(* CODESYS project CtaAppBmk_1.0.0.0.library
   Description: Bmk Library der CTA
   Version: 1.0.0.0
   Title: CtaAppBmk
   Author: SIS
   Company: CTA
   DocFormat: reStructuredText
   Placeholder: CtaAppBmk
   DefaultNamespace: CtaAppBmk
   CompiledLibraryCompatibilityVersion: CODESYS V3.5 SP16 Patch 3
   LanguageModelAttribute: qualified-access-only

Project tree, tasks and I/O mapping:
  libraries: CtaSysBase, 1.0.0.0 (CTA); TextListUtils, * (System); CtaVisSymbols, 1.0.0.0 (CTA); VisuSymbols, 4.5.0.0 (System)
  40 Visualizations/
    visualisation visObjInfoIntern
    visualisation visObjInfo
  30 Program Organization Units/
    function block fbBMK [ST]: proGetBMK, proGetAKS, proGetVendorDesignation, proGetCustomerDesignation, proGetObjectId, proNoBmkInList
  00000000-0000-0000-0000-000000000000|D:\CoDeSys\LibrariesV3\trunk\Intern\CAA\CAA Template\3.4.0.0 draft\Placeholder.xml
  00000000-0000-0000-0000-000000000000|D:\CoDeSys\LibrariesV3\trunk\Intern\CAA\CAA Template\3.2.0.3 draft\Prefix.pdf
  00000000-0000-0000-0000-000000000000|D:\CoDeSys\LibrariesV3\trunk\Intern\CAA\CAA Template\3.5.2.0 draft\Placeholder.xml
  20 Structs/
  50 Images/
  10 Documenation/
    global variables VersionHistory
    global variables readMe
  21 Interface/
    interface ITF_BMK: proGetAKS, proGetBMK, proGetObjectId, proNoBmkInList, proGetCustomerDesignation, proGetVendorDesignation
  11 Library Parameter/
    global variables Parameter
  12 Konstanten/
  60 Textlisten/
  13 Globale Variablen/
  text list GlobalTextList
*)

// 10 Documenation/VersionHistory
(* 

.. image:: ../../Images/CTA_Logo.jpg
   :align: right
   :width: 15% 

**Vorlage**   


============ =========== =========== ============================================
**Date**     **Version** **Author**  **Change**
------------ ----------- ----------- --------------------------------------------
04.03.2021   0.0.0.0     SIS         Vorlage erstellt

============ =========== =========== ============================================


*)
VAR_GLOBAL
    stInfo : STRING:= '0.0.0.0, Vorlage, CTA';
END_VAR

// 10 Documenation/readMe
(*

**ReadMe**
 
 |	**Empfehlung**
 |
 |	Dokumentrieren Sie die Library für eine nachhaltige Entwicklung
 |     
 | *Beispiel* 
 |
 | Dies ist die Vorlage Library der CTA. Erstellen Sie ihre Library anhand dieser Vorlage.
*)

VAR_GLOBAL
    xReadMeDone              :   BOOL;
END_VAR

// 11 Library Parameter/Parameter
{attribute 'qualified_only' := ''}
VAR_GLOBAL CONSTANT
	stTextListBmk					: STRING := 'BMK';
	stTextListAks					: STRING := 'AKS';
	stTextListVendorDesignation		: STRING := 'VendorDesignation';
	stTextListCustomerDesignation	: STRING := 'CustomerDesignation';
END_VAR

// 30 Program Organization Units/fbBMK
(* BMK Functionblock single Responsibility operating resources indicator BMK *)
{attribute 'enable_dynamic_creation'}
FUNCTION_BLOCK fbBMK EXTENDS CtaSysBase.fbBASE IMPLEMENTS ITF_BMK
VAR_INPUT
	/// Object ID
	{attribute 'monitoring_encoding' := 'UTF-8'}
	stObjId: STRING(20);
END_VAR
VAR
	/// Flag no BMK in List
	xNoBmkInList: BOOL;
END_VAR

{IF NOT defined (task:VISU_TASK) AND (defined (task:PLC_Task) OR defined (resource:Steuerung))}
    {error 'No VisualizationManager or No VISU_TASK in Application'}  
{END_IF}

{attribute 'monitoring':='call'}
{attribute 'monitoring_encoding' := 'UTF-8'}
PROPERTY proGetBMK : STRING(7)
GET
proGetBMK := '';
IF stObjId <> '' THEN
	(*Language dependent text*)
	TLU.GetText(Parameter.stTextListBmk,stObjId,ADR(proGetBMK),SIZEOF(proGetBMK));
	(* Set xNoBmkInList if no BMK is found*)
	IF proGetBMK = '' THEN
		xNoBmkInList := TRUE;
        proGetBMK    := '-';
	ELSE
		xNoBmkInList := FALSE;
	END_IF;
ELSE
    proGetBMK    := '-';    
END_IF;
END_GET
END_PROPERTY

{attribute 'monitoring':='call'}
{attribute 'monitoring_encoding' := 'UTF-8'}
PROPERTY proGetAKS : STRING(40)
GET
proGetAKS := '';
IF stObjId <> '' THEN
	(*Language dependent text*)
	TLU.GetText(Parameter.stTextListAks,stObjId,ADR(proGetAKS),SIZEOF(proGetAKS));
END_IF;
END_GET
END_PROPERTY

{attribute 'monitoring':='call'}
{attribute 'monitoring_encoding' := 'UTF-8'}
PROPERTY proGetVendorDesignation : STRING(140)
GET
proGetVendorDesignation := '';
IF stObjId <> '' THEN
	(*Language dependent text*)
	TLU.GetText(Parameter.stTextListVendorDesignation,stObjId,ADR(proGetVendorDesignation),SIZEOF(proGetVendorDesignation)); 
    IF proGetVendorDesignation = '' THEN
        proGetVendorDesignation := proGetInstancePath;
	END_IF;
ELSE
    proGetVendorDesignation := proGetInstancePath;    
END_IF;
END_GET
END_PROPERTY

{attribute 'monitoring':='call'}
{attribute 'monitoring_encoding' := 'UTF-8'}
PROPERTY proGetCustomerDesignation : STRING(100)
GET
VAR
    dwState :   DWORD;
END_VAR
proGetCustomerDesignation := '';
IF stObjId <> '' THEN
	(*Language dependent text*)
	__TRY
		dwState := TLU.GetText(Parameter.stTextListCustomerDesignation,stObjId,ADR(proGetCustomerDesignation),SIZEOF(proGetCustomerDesignation));
	__CATCH
		proGetCustomerDesignation := '';
	__ENDTRY	
END_IF;
END_GET
END_PROPERTY

{attribute 'monitoring':='call'}
{attribute 'monitoring_encoding' := 'UTF-8'}
PROPERTY proGetObjectId : STRING(20)
GET
proGetObjectId := stObjId;
END_GET
END_PROPERTY

{attribute 'monitoring':='call'}
{attribute 'monitoring_encoding' := 'UTF-8'}
PROPERTY proNoBmkInList : BOOL
GET
VAR
	stTestBMK :	STRING(7);
END_VAR
IF stObjId <> '' THEN
	(*Get state of xNoBmkInList*)
	stTestBMK := proGetBMK;
	proNoBmkInList := xNoBmkInList;
END_IF;
END_GET
END_PROPERTY

END_FUNCTION_BLOCK

// 21 Interface/ITF_BMK
/// BMK Interface single Responsibility operating resources indicator BMK
INTERFACE ITF_BMK EXTENDS CtaSysBase.ITF_BASE

{attribute 'monitoring':='call'}
PROPERTY proGetAKS : STRING(40)
GET
END_GET
END_PROPERTY

{attribute 'monitoring':='call'}
PROPERTY proGetBMK : STRING(7)
GET
END_GET
END_PROPERTY

{attribute 'monitoring':='call'}
PROPERTY proGetObjectId : STRING(20)
GET
END_GET
END_PROPERTY

{attribute 'monitoring':='call'}
PROPERTY proNoBmkInList : BOOL
GET
END_GET
END_PROPERTY

{attribute 'monitoring':='call'}
PROPERTY proGetCustomerDesignation : STRING(100)
GET
END_GET
END_PROPERTY

{attribute 'monitoring':='call'}
PROPERTY proGetVendorDesignation : STRING(140)
GET
END_GET
END_PROPERTY

END_INTERFACE

// 40 Visualizations/visObjInfoIntern
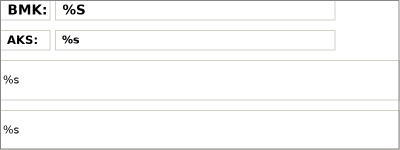
VISUALIZATION visObjInfoIntern  // 400x150
VAR_INPUT
	ITF_BMK_IN : ITF_BMK;
END_VAR
    Textfield (0,0 50x20), "BMK:"
    Textfield (0,30 50x20), "AKS:", invisible if: ITF_BMK_IN.proGetAKS = ''
    Textfield (55,0 280x20), "%S", text variable: SEL(ITF_BMK_IN.proNoBmkInList,ITF_BMK_IN.proGetBMK,'No BMK Found')
    Textfield (55,30 280x20), "%s", text variable: ITF_BMK_IN.proGetAKS, invisible if: ITF_BMK_IN.proGetAKS = ''
    Textfield (0,60 400x40), "%s", tooltip "Hersteller Bezeichnung", text variable: ITF_BMK_IN.proGetVendorDesignation, invisible if: ITF_BMK_IN.proGetVendorDesignation = ''
    Textfield (0,110 400x40), "%s", tooltip "Kunden Bezeichnung", text variable: ITF_BMK_IN.proGetCustomerDesignation, invisible if: ITF_BMK_IN.proGetCustomerDesignation = ''
END_VISUALIZATION

// 40 Visualizations/visObjInfo
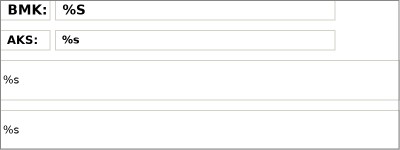
VISUALIZATION visObjInfo  // 400x150
VAR_INPUT
	ITF_BMK_IN : ITF_BMK;
END_VAR
    Frame (0,0 400x150), invisible if: ITF_BMK_IN =0
        shows visObjInfoIntern(ITF_BMK_IN := ITF_BMK_IN)
END_VISUALIZATION
